// SIMATIC S7-200 project (STEP 7-Micro/WIN), CPU 224XP REL 02.01

ORGANIZATION_BLOCK MAIN:OB1
TITLE=PROGRAM COMMENTS
BEGIN
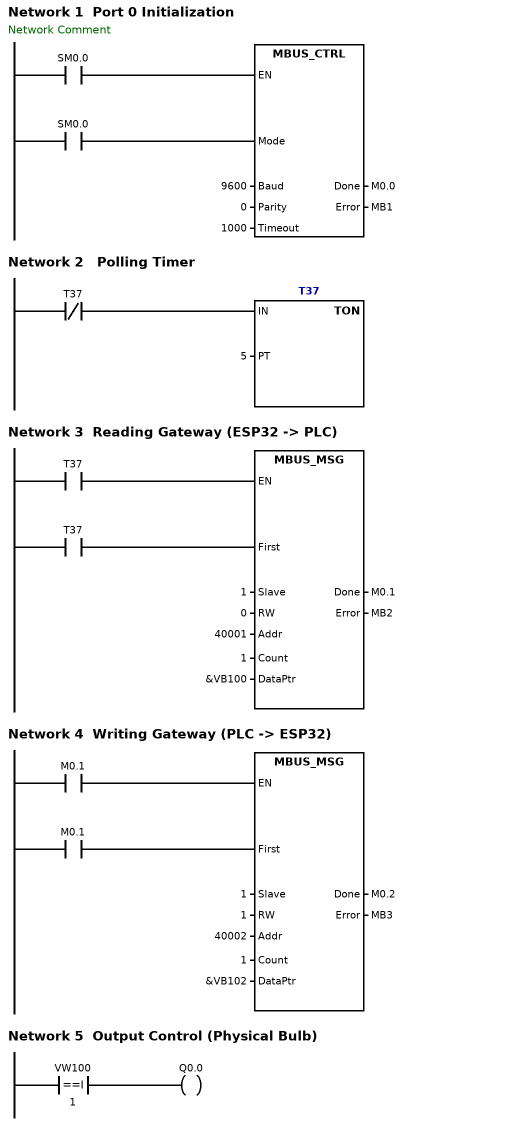
Network 1 // Port 0 Initialization
// Network Comment
LD     SM0.0
=      L60.0
LD     SM0.0
=      L63.7
LD     L60.0
CALL   MBUS_CTRL:SBR1, L63.7, 9600, 0, 1000, M0.0, MB1
Network 2 //  Polling Timer
LDN    T37
TON    T37, 5
Network 3 // Reading Gateway (ESP32 -> PLC)
LD     T37
=      L60.0
LD     T37
=      L63.7
LD     L60.0
CALL   MBUS_MSG:SBR2, L63.7, 1, 0, 40001, 1, &VB100, M0.1, MB2
Network 4 // Writing Gateway (PLC -> ESP32)
LD     M0.1
=      L60.0
LD     M0.1
=      L63.7
LD     L60.0
CALL   MBUS_MSG:SBR2, L63.7, 1, 1, 40002, 1, &VB102, M0.2, MB3
Network 5 // Output Control (Physical Bulb)
LDW=   VW100, 1
=      Q0.0
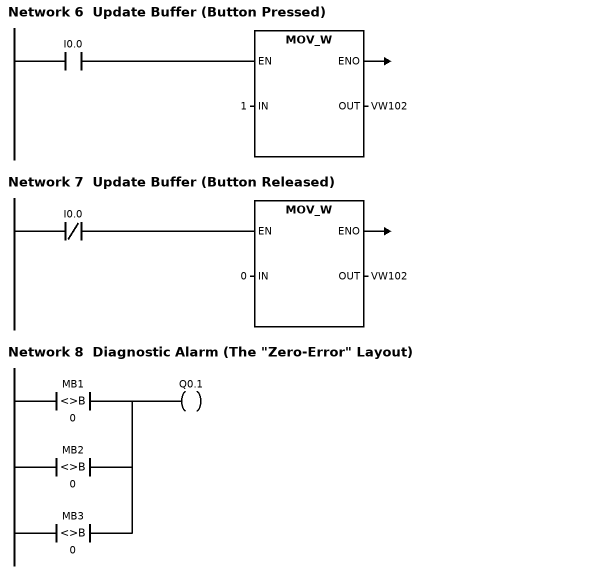
Network 6 // Update Buffer (Button Pressed)
LD     I0.0
MOVW   1, VW102
Network 7 // Update Buffer (Button Released)
LDN    I0.0
MOVW   0, VW102
Network 8 // Diagnostic Alarm (The "Zero-Error" Layout)
LDB<>  MB1, 0
OB<>   MB2, 0
OB<>   MB3, 0
=      Q0.1
END_ORGANIZATION_BLOCK

// SBR1: protected block, not included

// SBR2: protected block, not included

// SBR3: protected block, not included
